{attribute 'qualified_only'}
VAR_GLOBAL
	bLampeGruen		:	BOOL;
	bLampeGelb		:	BOOL;
	bLampeRot		:	BOOL;
	
	bSchalterBlau	:	BOOL;
	bSchalterGelb	:	BOOL;
END_VAR

(* stored: Version 1.1.0.1, ProductVersion 3.1.4024.12
   GVL I0: Id {7c3048ef-f548-42be-bc03-806430738406} *)
